FUNCTION_BLOCK MUX_ADC
VAR_INPUT
	CLK : BOOL;
	ADC_INPUT : INT;
END_VAR
VAR_OUTPUT
	SELLECT : ARRAY[0..4] OF BOOL;
	ADC_OUTPUT : ARRAY[0..31] OF INT;
END_VAR
VAR
	
	CNT_MUX : UINT;	
	PREV_CLK : BOOL;
	CS : ARRAY[0..4] OF BOOL;
	ADC_TEMP : ARRAY[0..31] OF INT;

END_VAR

SELLECT := CS;
ADC_OUTPUT := ADC_TEMP;


IF (PREV_CLK=FALSE AND CLK=TRUE) THEN
	
	ADC_TEMP[CNT_MUX] := ADC_INPUT;	

	CNT_MUX := CNT_MUX + 1;
	IF CNT_MUX > 31 THEN
		CNT_MUX := 0;
	END_IF
	
	CS[0] := UINT_TO_BOOL(CNT_MUX AND 16#01);
	CS[1] := UINT_TO_BOOL(CNT_MUX AND 16#02);
	CS[2] := UINT_TO_BOOL(CNT_MUX AND 16#04);
	CS[3] := UINT_TO_BOOL(CNT_MUX AND 16#08);
	CS[4] := UINT_TO_BOOL(CNT_MUX AND 16#10);
	
	
END_IF 

PREV_CLK := CLK;

END_FUNCTION_BLOCK

(* stored: Version 1.1.0.1, ProductVersion 3.1.4024.12
   POU MUX_ADC: Id {6e85e4dd-135c-4c09-af67-d0b75cdc18aa}, SpecialFunc None *)
